FUNCTION_BLOCK fbAxisPosCtrl
VAR_INPUT

	bAxis1EN : BOOL;
	bAxis2EN : BOOL;
	bAxis3EN : BOOL;
	bAxis4EN : BOOL;

	bPosStart : BOOL;
	bHomingRdy : BOOL;
	wTargetPosNum : DWORD;
	lrFixVelo : LREAL;
	lrFixAcc : LREAL;
	lrFixDcc : LREAL;
	lrCurrentServoPos : LREAL;
	lrPos1 : LREAL;
	lrPos2 : LREAL;
	lrPos3 : LREAL;
	lrPos4 : LREAL;
	lrPos5 : LREAL;
	lrPos6 : LREAL;
	lrPos7 : LREAL;
	lrPos8 : LREAL;
	lrPos9 : LREAL;
	lrPos10 : LREAL;
	lrPos11 : LREAL;
	lrPos12 : LREAL;
	lrPos13 : LREAL;
	lrPos14 : LREAL;
	lrPos15 : LREAL;
	lrPos16 : LREAL;
	lrPos17 : LREAL;
	lrPos18 : LREAL;
	lrPos19 : LREAL;
	lrPos20 : LREAL;
	lrPos21 : LREAL;
	lrPos22 : LREAL;
	lrPos23 : LREAL;
	lrPos24 : LREAL;
	lrPos25 : LREAL;

END_VAR
VAR_IN_OUT
	Arm1HorzReady: BOOL;
	Arm1VertReady: BOOL;
	Arm1Vert : axis_ref;
	Arm1Horz : axis_ref;
END_VAR

VAR_OUTPUT

	AxisStopEn : BOOL;

END_VAR
VAR
	Stoptimer: TON;
	AxisStopbit: BOOL;
	TimerMove: TON;
	BlockStartBit: BOOL;
	PosSV: LREAL;
	Move1: BOOL;
	Move2: BOOL;
	Move3: BOOL;
	Move4: BOOL;
	Move5: BOOL;
	Move6: BOOL;
	Move7: BOOL;
	Move8: BOOL;
	Move9: BOOL;
	Move10: BOOL;
	Move11: BOOL;
	Move12: BOOL;
	Move13: BOOL;
	Move14: BOOL;
	Move15: BOOL;
	Move16: BOOL;
	Move17: BOOL;
	Move18: BOOL;
	Move19: BOOL;
	Move20: BOOL;
	Move21: BOOL;
	Move22: BOOL;
	Move23: BOOL;
	Move24: BOOL;
	Move25: BOOL;
	Halt1: MC_Halt;
	Halt2: MC_Halt;
	Halt3: MC_Halt;
	Halt4: MC_Halt;
	ArmMoveTostation2: MC_MoveAbsolute;
	ArmMoveTostation: MC_MoveAbsolute;
	ArmMoveTostation3: MC_MoveAbsolute;
	ArmMoveTostation4: MC_MoveAbsolute;
	AxisStopEn1: BOOL;
	AxisStopEn2: BOOL;
	AxisStopEn3: BOOL;
	AxisStopEn4: BOOL;
	Arm1VertReadStatus: MC_ReadStatus;
	Arm1HorzReadStatus: MC_ReadStatus;
END_VAR
VAR // added by the converter: edge detectors and wires of the graphical bodies
    _w1, _w2, _w3, _w4, _w5, _w6, _w7, _w8, _w9, _w10, _w11, _w12, _w13, _w14, _w15, _w16, _w17, _w18, _w19, _w20, _w21, _w22, _w23, _w24, _w25 : LREAL;
END_VAR

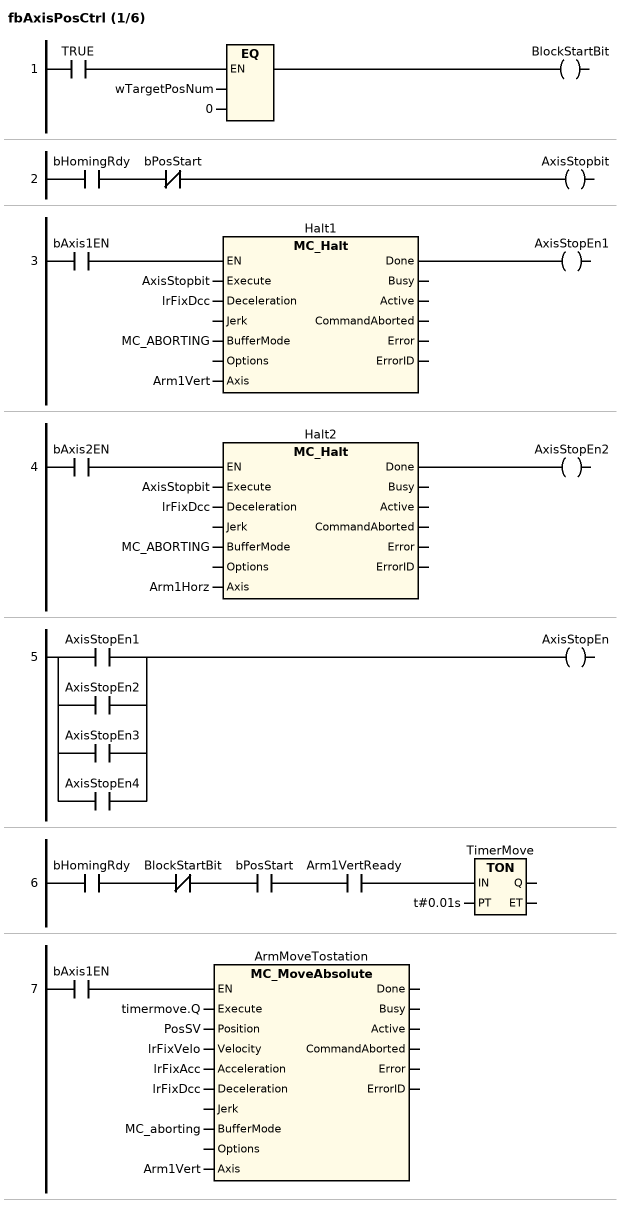
// NETWORK 1
BlockStartBit := wTargetPosNum = 0;

// NETWORK 2
AxisStopbit := bHomingRdy AND NOT bPosStart;

// NETWORK 3
IF bAxis1EN THEN
    Halt1(Execute := AxisStopbit, Deceleration := lrFixDcc, BufferMode := MC_ABORTING, Axis := Arm1Vert); // MC_Halt
END_IF
AxisStopEn1 := Halt1.Done;

// NETWORK 4
IF bAxis2EN THEN
    Halt2(Execute := AxisStopbit, Deceleration := lrFixDcc, BufferMode := MC_ABORTING, Axis := Arm1Horz); // MC_Halt
END_IF
AxisStopEn2 := Halt2.Done;

// NETWORK 5
AxisStopEn := AxisStopEn1 OR AxisStopEn2 OR AxisStopEn3 OR AxisStopEn4;

// NETWORK 6
TimerMove(IN := bHomingRdy AND NOT BlockStartBit AND bPosStart AND Arm1VertReady, PT := t#0.01s); // TON

// NETWORK 7
IF bAxis1EN THEN
    ArmMoveTostation(
        Execute := timermove.Q,
        Position := PosSV,
        Velocity := lrFixVelo,
        Acceleration := lrFixAcc,
        Deceleration := lrFixDcc,
        BufferMode := MC_aborting,
        Axis := Arm1Vert); // MC_MoveAbsolute
END_IF

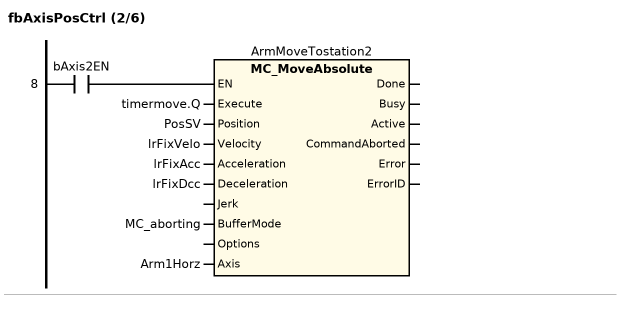
// NETWORK 8
IF bAxis2EN THEN
    ArmMoveTostation2(
        Execute := timermove.Q,
        Position := PosSV,
        Velocity := lrFixVelo,
        Acceleration := lrFixAcc,
        Deceleration := lrFixDcc,
        BufferMode := MC_aborting,
        Axis := Arm1Horz); // MC_MoveAbsolute
END_IF

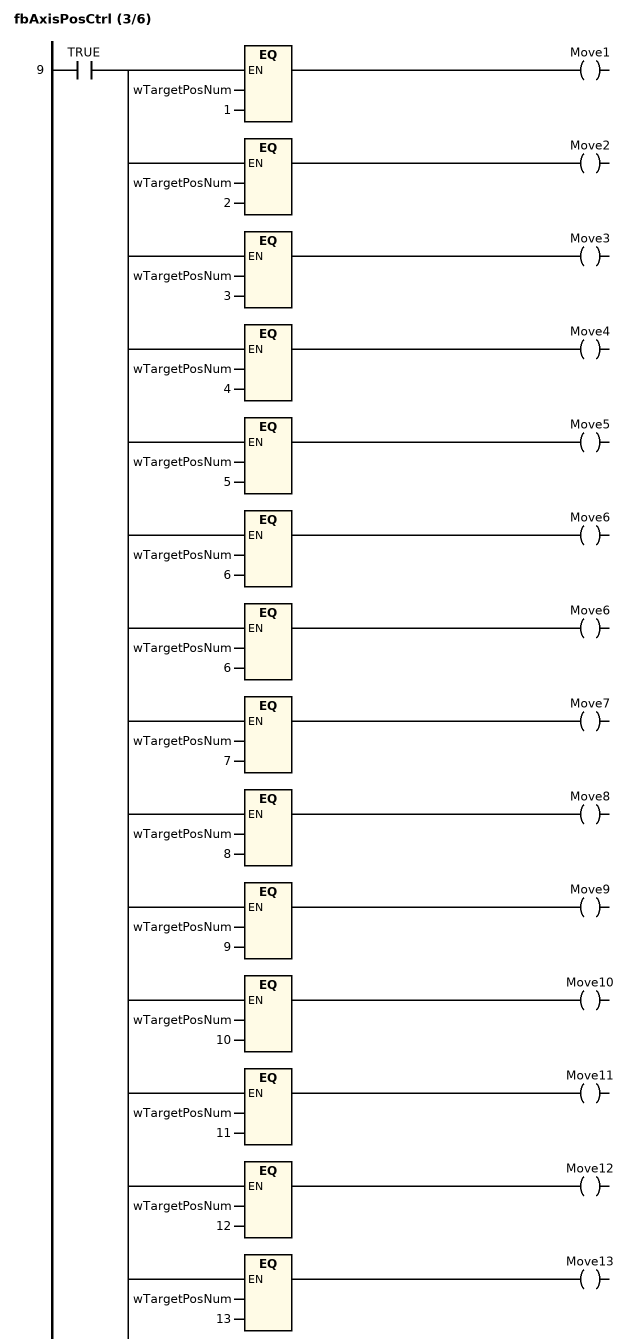
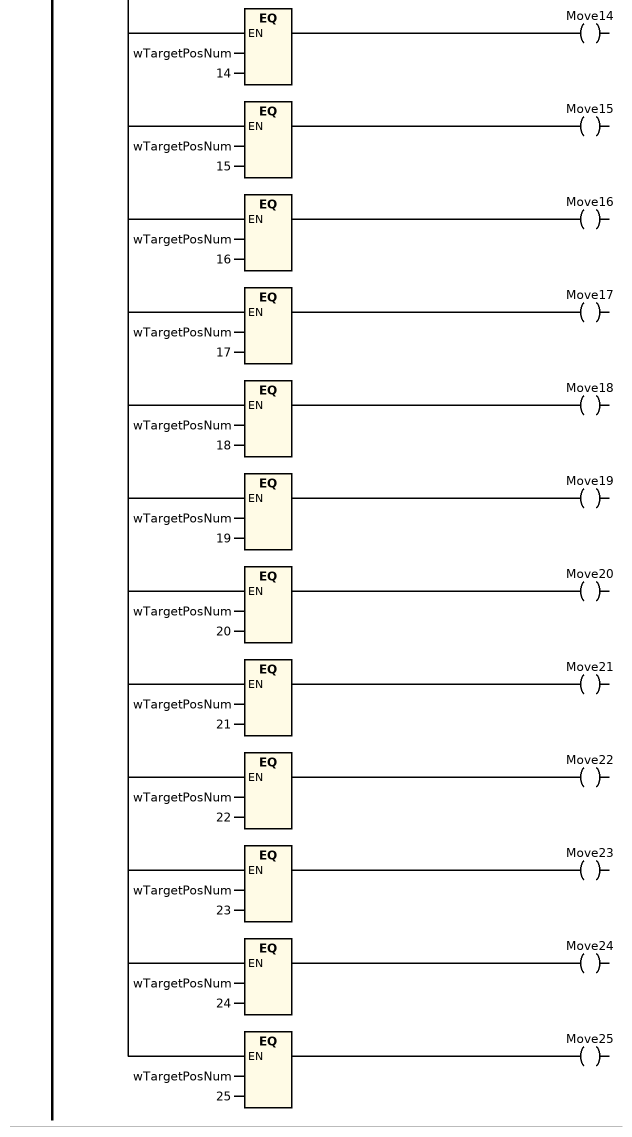
// NETWORK 9
Move1 := wTargetPosNum = 1;
Move2 := wTargetPosNum = 2;
Move3 := wTargetPosNum = 3;
Move4 := wTargetPosNum = 4;
Move5 := wTargetPosNum = 5;
Move6 := wTargetPosNum = 6;
Move6 := wTargetPosNum = 6;
Move7 := wTargetPosNum = 7;
Move8 := wTargetPosNum = 8;
Move9 := wTargetPosNum = 9;
Move10 := wTargetPosNum = 10;
Move11 := wTargetPosNum = 11;
Move12 := wTargetPosNum = 12;
Move13 := wTargetPosNum = 13;
Move14 := wTargetPosNum = 14;
Move15 := wTargetPosNum = 15;
Move16 := wTargetPosNum = 16;
Move17 := wTargetPosNum = 17;
Move18 := wTargetPosNum = 18;
Move19 := wTargetPosNum = 19;
Move20 := wTargetPosNum = 20;
Move21 := wTargetPosNum = 21;
Move22 := wTargetPosNum = 22;
Move23 := wTargetPosNum = 23;
Move24 := wTargetPosNum = 24;
Move25 := wTargetPosNum = 25;

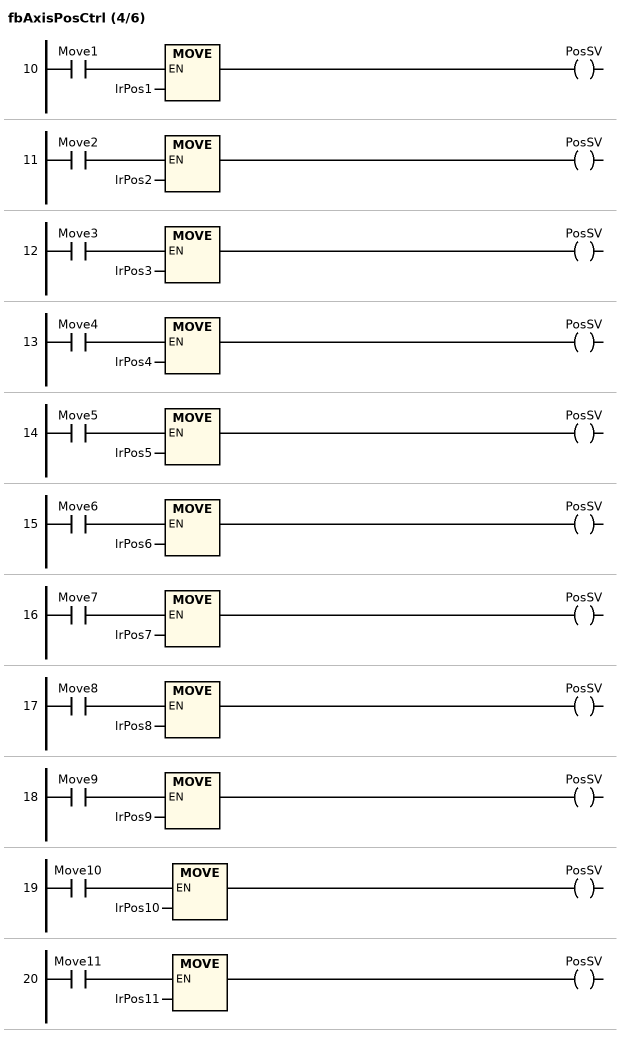
// NETWORK 10
IF Move1 THEN _w1 := lrPos1; END_IF
PosSV := _w1;

// NETWORK 11
IF Move2 THEN _w2 := lrPos2; END_IF
PosSV := _w2;

// NETWORK 12
IF Move3 THEN _w3 := lrPos3; END_IF
PosSV := _w3;

// NETWORK 13
IF Move4 THEN _w4 := lrPos4; END_IF
PosSV := _w4;

// NETWORK 14
IF Move5 THEN _w5 := lrPos5; END_IF
PosSV := _w5;

// NETWORK 15
IF Move6 THEN _w6 := lrPos6; END_IF
PosSV := _w6;

// NETWORK 16
IF Move7 THEN _w7 := lrPos7; END_IF
PosSV := _w7;

// NETWORK 17
IF Move8 THEN _w8 := lrPos8; END_IF
PosSV := _w8;

// NETWORK 18
IF Move9 THEN _w9 := lrPos9; END_IF
PosSV := _w9;

// NETWORK 19
IF Move10 THEN _w10 := lrPos10; END_IF
PosSV := _w10;

// NETWORK 20
IF Move11 THEN _w11 := lrPos11; END_IF
PosSV := _w11;

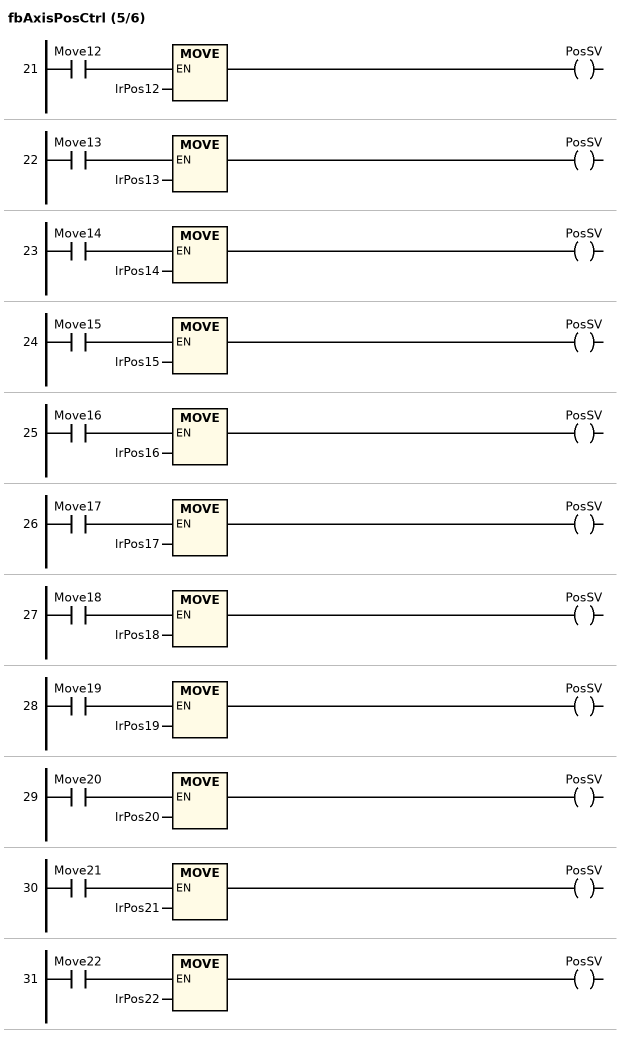
// NETWORK 21
IF Move12 THEN _w12 := lrPos12; END_IF
PosSV := _w12;

// NETWORK 22
IF Move13 THEN _w13 := lrPos13; END_IF
PosSV := _w13;

// NETWORK 23
IF Move14 THEN _w14 := lrPos14; END_IF
PosSV := _w14;

// NETWORK 24
IF Move15 THEN _w15 := lrPos15; END_IF
PosSV := _w15;

// NETWORK 25
IF Move16 THEN _w16 := lrPos16; END_IF
PosSV := _w16;

// NETWORK 26
IF Move17 THEN _w17 := lrPos17; END_IF
PosSV := _w17;

// NETWORK 27
IF Move18 THEN _w18 := lrPos18; END_IF
PosSV := _w18;

// NETWORK 28
IF Move19 THEN _w19 := lrPos19; END_IF
PosSV := _w19;

// NETWORK 29
IF Move20 THEN _w20 := lrPos20; END_IF
PosSV := _w20;

// NETWORK 30
IF Move21 THEN _w21 := lrPos21; END_IF
PosSV := _w21;

// NETWORK 31
IF Move22 THEN _w22 := lrPos22; END_IF
PosSV := _w22;

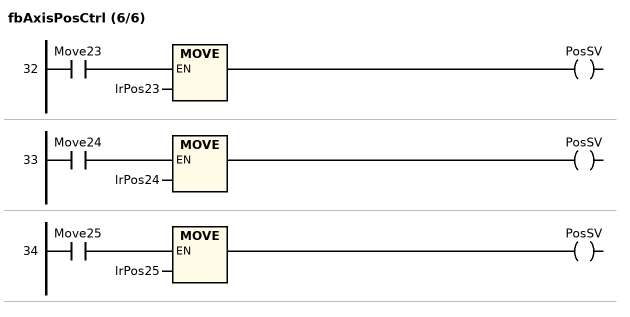
// NETWORK 32
IF Move23 THEN _w23 := lrPos23; END_IF
PosSV := _w23;

// NETWORK 33
IF Move24 THEN _w24 := lrPos24; END_IF
PosSV := _w24;

// NETWORK 34
IF Move25 THEN _w25 := lrPos25; END_IF
PosSV := _w25;

END_FUNCTION_BLOCK

(* stored: Version 1.1.0.1, ProductVersion 3.1.4024.12
   POU fbAxisPosCtrl: Id {16ad2995-58fe-4247-b766-770c9fde1859}, SpecialFunc None *)
